{attribute 'pack_mode' := '1'}
TYPE ST_3002_Supervisor_Status EXTENDS ST_SupervisorHeader:
	STRUCT
		Status			   : E_3002_Status := E_3002_Status.Ok;
		Set_Estop		   : E_3002_Set_ESTOP;
		{attribute 'hide'}
		Number_of_sections : UINT := 0;
		//Section_IDs		   : ARRAY[0..0] OF UINT := [1];//List of sections to send in the response message 3102
	END_STRUCT
END_TYPE

(* stored: Version 1.1.0.1, ProductVersion 3.1.4026.17
   DUT ST_3002_Supervisor_Status: Id {7b244444-4475-46b5-8f8f-90546fc15de9} *)
